INTERFACE I_PackMLMode

END_INTERFACE

(* stored: Version 1.1.0.1, ProductVersion 3.1.4024.12
   Itf I_PackMLMode: Id {c750d27f-ab1f-4fed-bfa8-5dd2e8979068} *)
